{attribute addProperty BoxType "AX8118-0000-0102-0102"}
{attribute addProperty Id "DeviceDevice_F82A60211620Ch_ACh_A_B17182A2176220WcStateAT %I*WcState_F855686C1620InfoDataAT %I*InfoData_F030DC9B200250"}
{attribute addProperty CRC "4187634827"}
{attribute addProperty SizeInBites "408"}
{attribute addProperty SizeInBytes "51"}
TYPE AX8118_3F1F35B3 :
STRUCT
	{attribute addProperty Name "Device"}
	Device : Device_F82A6021;
	{attribute addProperty Name "Ch_A"}
	Ch_A : Ch_A_B17182A2;
	{attribute addProperty Name "WcState"}
	WcState : WcState_F855686C;
	{attribute addProperty Name "InfoData"}
	InfoData : InfoData_F030DC9B;
END_STRUCT
END_TYPE

(* stored: Version 1.2.0.0, ProductVersion 3.1.4024.9
   DUT AX8118_3F1F35B3: Id {b8d3d37a-1474-4c69-a895-7443ec7f9f48} *)
